TYPE ExampleDomain_Priv :
STRUCT
	smgr					: I_StateManager;
END_STRUCT
END_TYPE

(* stored: Version 1.1.0.1
   DUT ExampleDomain_Priv: Id {b5879e2d-3173-4d3f-bd19-ed68ec7cecd1} *)
